ABB RobotStudio station: robot2gyak.rspag

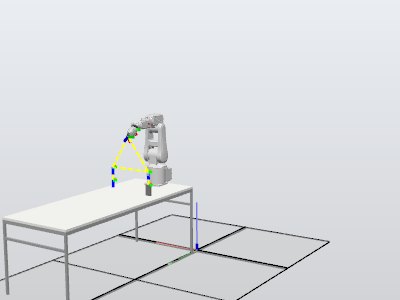
--- station ---
Station robot2gyak (saved by RobotStudio 25.3.11371.0)
Controller IRB120_3_58__01, task T_ROB1: task frame (RAPID world) sits at (345.97, 203.99, 678.76) mm, rotated rx 0 ry 0 rz 92.79 deg in the station
Controller IRB120_3_58__01
  mechanical unit ROB_1: IRB120_3_58__01, 6 joints, base frame (0, 0, 0) mm
Layout (positions relative to the parent item):
  - table [part, from D:\Table.rslib] at (-7.18, 83.56, 675.03) mm
  - IRB120_3_58__01 [mechanism, from %ABB.RobotStudio.Models.IRB120%\IRB120_3_58_G_01.rslib] at (345.97, 203.99, 678.76) mm, rotated rx 0 ry 0 rz 92.79 deg; joint values [0, 0, 0, 0, 0.5236, 0] (rad or m)
  - Part_1 [part] at (107.24, 605.1, 675.03) mm, size 50 x 25 x 100 mm
  - Smart_Gripper_Servo_Fingers [mechanism, from %ABB.RobotStudio.Models.SmartGripper%\ABB_Smart_Gripper_Servo_Fingers.rslib] at (328.22, 567.91, 1272.76) mm, rotated rx 180 ry 60 rz -87.21 deg; joint values [0.0125] (rad or m)
  - SmartComponent_1 [smart component]
      signals: DI OpenClose
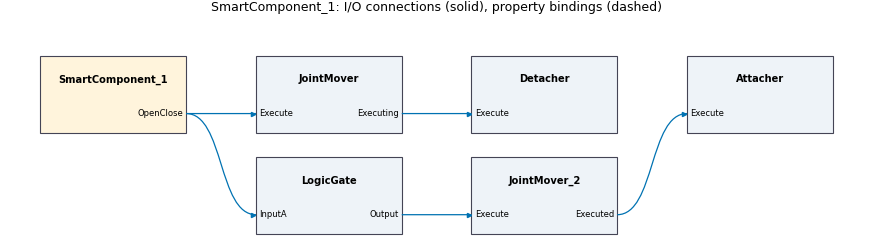
      connections:
        SmartComponent_1.OpenClose -> JointMover.Execute
        JointMover.Executing -> Detacher.Execute
        SmartComponent_1.OpenClose -> LogicGate.InputA
        LogicGate.Output -> JointMover_2.Execute
        JointMover_2.Executed -> Attacher.Execute
    - Attacher [smart component, from Components\Attacher.rslib]
        properties: Parent=Smart_Gripper_Servo_Fingers; Flange=0; Child=Part_1; Mount=false; Offset=[0 0 0]; Orientation=[0 0 0]
    - Detacher [smart component, from Components\Detacher.rslib]
        properties: Child=Part_1; KeepPosition=true
    - JointMover [smart component, from Components\JointMover.rslib]
        properties: Mechanism=Smart_Gripper_Servo_Fingers; Relative=false; Duration=2; J1=0.025
    - JointMover_2 [smart component, from Components\JointMover.rslib]
        properties: Mechanism=Smart_Gripper_Servo_Fingers; Relative=false; Duration=0; J1=0.0125
    - LogicGate [smart component, from Components\LogicGate.rslib]
        properties: Operator=NOT; Delay=0
Attachment: Smart_Gripper_Servo_Fingers is attached to IRB120_3_58__01 / Link6
Attachment: Part_1 is attached to Smart_Gripper_Servo_Fingers / HandBase
Station logic (signal -> signal, property => property):
  IRB120_3_58__01.Hand -> SmartComponent_1.OpenClose

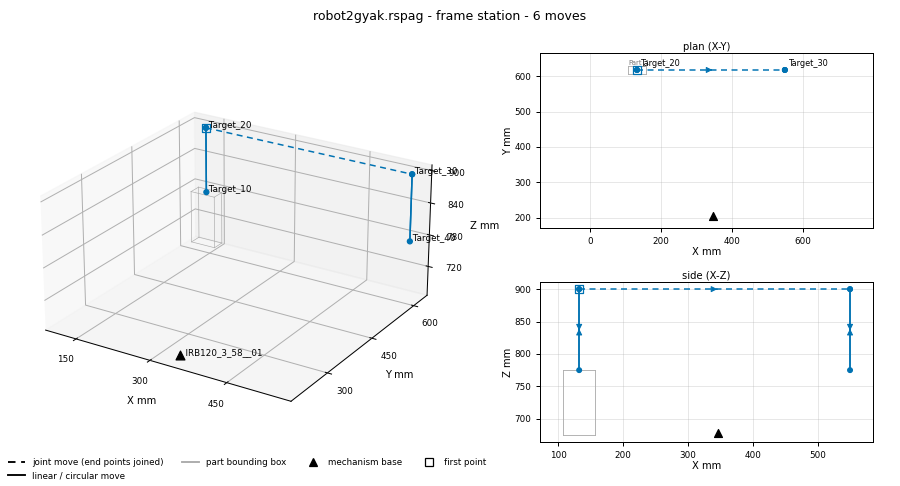
[picture p0: tool path of robot2gyak.rspag in frame station, 6 of 8 moves have a stored position in this frame; points joined in program order, loops and branches not executed]
--- Controller Data/IRB120_3_58__01/RAPID/TASK1/PROGMOD/CalibData.mod ---
MODULE CalibData
    PERS tooldata Servo:=[TRUE,[[0,0,114.2],[1,0,0,0]],[0.215,[8.7,12.3,49.2],[1,0,0,0],0.00021,0.00024,0.00009]];
ENDMODULE

--- Controller Data/IRB120_3_58__01/RAPID/TASK1/PROGMOD/Module1.mod ---
MODULE Module1
    CONST jointtarget Home:=[[0,0,0,0,30,0],[9E+09,9E+09,9E+09,9E+09,9E+09,9E+09]];
    CONST robtarget Target_20:=[[423.533315766,193.317682913,221.237328747],[0,0.024377531,0.999702824,0],[0,0,0,0],[9E+09,9E+09,9E+09,9E+09,9E+09,9E+09]];
    CONST robtarget Target_10:=[[423.533315766,193.317682913,96.268328747],[0,0.024377531,0.999702824,0],[0,0,0,0],[9E+09,9E+09,9E+09,9E+09,9E+09,9E+09]];
    CONST robtarget Target_30:=[[403.171600029,-223.942801174,221.237328747],[0,0.024377531,0.999702824,0],[-1,0,-1,0],[9E+09,9E+09,9E+09,9E+09,9E+09,9E+09]];
    CONST robtarget Target_40:=[[403.171600029,-223.942801174,96.268328747],[0,0.024377531,0.999702824,0],[-1,0,-1,0],[9E+09,9E+09,9E+09,9E+09,9E+09,9E+09]];
    !***********************************************************
    !
    ! Module:  Module1
    !
    ! Description:
    !   <Insert description here>
    !
    ! Author: anlal
    !
    ! Version: 1.0
    !
    !***********************************************************


    !***********************************************************
    !
    ! Procedure main
    !
    !   This is the entry point of your program
    !
    !***********************************************************
    PROC main()
        Path_10;
    ENDPROC
    PROC Path_10()
        SetDO Hand, 1;
        WaitTime 2;
        MoveAbsJ Home,v1000,z0,Servo\WObj:=wobj0;
        MoveJ Target_20,v1000,z100,Servo\WObj:=wobj0;
        MoveL Target_10,v1000,fine,Servo\WObj:=wobj0;
        SetDO Hand, 0;
        WaitTime 2;
        MoveL Target_20,v1000,z100,Servo\WObj:=wobj0;
        MoveJ Target_30,v1000,z100,Servo\WObj:=wobj0;
        MoveL Target_40,v1000,fine,Servo\WObj:=wobj0;
        SetDO Hand, 1;
        WaitTime 2;
        MoveL Target_30,v1000,z100,Servo\WObj:=wobj0;
        MoveAbsJ Home,v1000,z0,Servo\WObj:=wobj0;
    ENDPROC
ENDMODULE

--- Controller Data/IRB120_3_58__01/SYSPAR/EIO.cfg ---
EIO:CFG_1.0:6:1::
#
ETHERNETIP_DEVICE:

      -Name "Local_IO" -VendorName "ABB Robotics" -ProductName "DSQC1030"\
      -Label "ABB Local I/O Device" -Address "192.168.125.3" -VendorId 75\
      -ProductCode 29 -DeviceType 12 -OutputAssembly 100 -InputAssembly 101\
      -ConfigurationAssembly 102 -InputConnectionType "POINT2POINT"\
      -ConnectionPriority "SCHEDULE" -OutputSize 2 -InputSize 2\
      -ConfigurationSize 8\
      -ConfigurationData00 "01 02 09 10 01 08 10 01 00 00 00 00 00 00 00 00"\
      -O2T_RPI 40000 -T2O_RPI 40000
#
EIO_SIGNAL:

      -Name "Hand" -SignalType "DO" -Device "Local_IO" -DeviceMap "1"
